// TIA Portal V20 export
FUNCTION_BLOCK "LER_SleepModeManager"   // FB184, LAD
// stored: Access Published, MemoryReserve 100, SetENOAutomatically false
   VAR_INPUT
      enable : Bool := TRUE;   // Enable sleep mode manager
      unitStatus : "LAF_typeUnitStatus";   // Unit status including stopped state and acknowledge command
      wakeUpReq : Bool;
      sleepDelay : Time;   // Idle time before sleep mode in minutes from HMI/recipe
      deepSleepDelay : Time;   // Time in sleep mode before deep sleep in minutes from HMI/recipe
   END_VAR
   VAR_OUTPUT
      sleepModeChangeReq : Bool;   // Request Unit mode change to sleep mode userMode02
      deepSleepModeChangeReq : Bool;   // Request Unit mode change to deep sleep mode userMode03
      wakeUpRecoveryRequired : Bool;
   END_VAR
   VAR
      instSleepDelay { ExternalAccessible := 'False'; ExternalVisible := 'False'; ExternalWritable := 'False'; S7_SetPoint := 'True'} : TON_TIME;
      instDeepSleepDelay { ExternalAccessible := 'False'; ExternalVisible := 'False'; ExternalWritable := 'False'; S7_SetPoint := 'True'} : TON_TIME;
      statStandbyReady { ExternalAccessible := 'False'; ExternalVisible := 'False'; ExternalWritable := 'False'} : Bool;
      statWakeUpRecoveryRequired { ExternalAccessible := 'False'; ExternalVisible := 'False'; ExternalWritable := 'False'} : Bool;
   END_VAR
   VAR_TEMP
      tempSleepDelayDone : Bool;
      tempDeepSleepDelayDone : Bool;
   END_VAR
   VAR CONSTANT
      MIN_TO_MS : LReal := 60000.0;   // Milliseconds per minute
      MAX_TIME_MIN : LReal := 35791.0;   // TIME max is about 24d20h31m23s
   END_VAR
BEGIN

REGION Network 1: Standby Ready
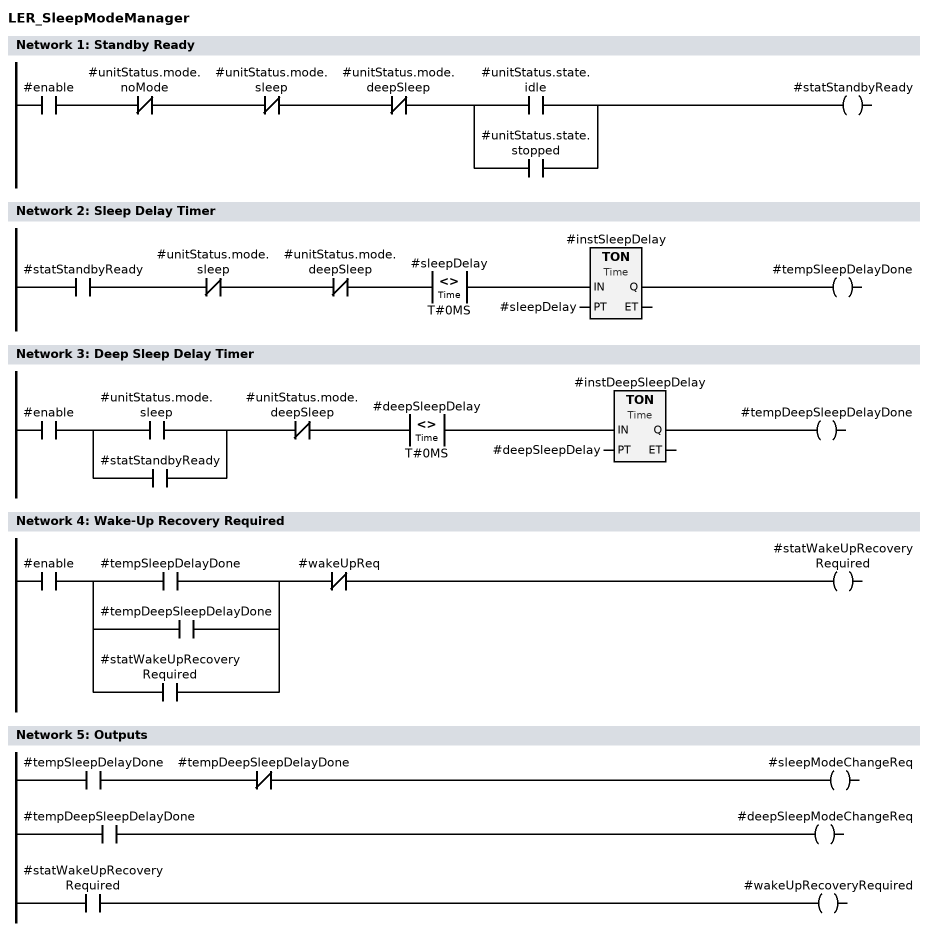
   RUNG wire#powerrail
      Contact( #enable )
      I_Contact( #unitStatus.mode.noMode )
      I_Contact( #unitStatus.mode.sleep )
      I_Contact( #unitStatus.mode.deepSleep )
      wire#w1
      Contact( #unitStatus.state.idle )
      wire#w2
      Coil( #statStandbyReady )
   END_RUNG
   RUNG wire#w1
      Contact( #unitStatus.state.stopped )
   END_RUNG wire#w2
   // the same network as SCL:
   #statStandbyReady := #enable AND NOT #unitStatus.mode.noMode AND NOT #unitStatus.mode.sleep AND NOT #unitStatus.mode.deepSleep AND (#unitStatus.state.idle OR #unitStatus.state.stopped);
END_REGION

REGION Network 2: Sleep Delay Timer
   RUNG wire#powerrail
      Contact( #statStandbyReady )
      I_Contact( #unitStatus.mode.sleep )
      I_Contact( #unitStatus.mode.deepSleep )
      { S7_Templates := "SrcType := Time" } NE_Contact(in1 := #sleepDelay, in2 := T#0MS)
      { S7_Templates := "time_type := Time" } #instSleepDelay.TON(pt := #sleepDelay, et =>)
      Coil( #tempSleepDelayDone )
   END_RUNG
   // the same network as SCL:
   #instSleepDelay(IN := #statStandbyReady AND NOT #unitStatus.mode.sleep AND NOT #unitStatus.mode.deepSleep AND (#sleepDelay <> T#0MS),   // TON
                   PT := #sleepDelay);
   #tempSleepDelayDone := #instSleepDelay.Q;
END_REGION

REGION Network 3: Deep Sleep Delay Timer
   RUNG wire#powerrail
      Contact( #enable )
      wire#w1
      Contact( #unitStatus.mode.sleep )
      wire#w2
      I_Contact( #unitStatus.mode.deepSleep )
      { S7_Templates := "SrcType := Time" } NE_Contact(in1 := #deepSleepDelay, in2 := T#0MS)
      { S7_Templates := "time_type := Time" } #instDeepSleepDelay.TON(pt := #deepSleepDelay, et =>)
      Coil( #tempDeepSleepDelayDone )
   END_RUNG
   RUNG wire#w1
      Contact( #statStandbyReady )
   END_RUNG wire#w2
   // the same network as SCL:
   #instDeepSleepDelay(IN := #enable AND (#unitStatus.mode.sleep OR #statStandbyReady) AND NOT #unitStatus.mode.deepSleep AND (#deepSleepDelay <> T#0MS),   // TON
                       PT := #deepSleepDelay);
   #tempDeepSleepDelayDone := #instDeepSleepDelay.Q;
END_REGION

REGION Network 4: Wake-Up Recovery Required
   RUNG wire#powerrail
      Contact( #enable )
      wire#w1
      Contact( #tempSleepDelayDone )
      wire#w2
      I_Contact( #wakeUpReq )
      Coil( #statWakeUpRecoveryRequired )
   END_RUNG
   RUNG wire#w1
      Contact( #tempDeepSleepDelayDone )
   END_RUNG wire#w2
   RUNG wire#w1
      Contact( #statWakeUpRecoveryRequired )
   END_RUNG wire#w2
   // the same network as SCL:
   #statWakeUpRecoveryRequired := #enable AND (#tempSleepDelayDone OR #tempDeepSleepDelayDone OR #statWakeUpRecoveryRequired) AND NOT #wakeUpReq;
END_REGION

REGION Network 5: Outputs
   RUNG wire#powerrail
      Contact( #tempSleepDelayDone )
      I_Contact( #tempDeepSleepDelayDone )
      Coil( #sleepModeChangeReq )
   END_RUNG
   RUNG wire#powerrail
      Contact( #tempDeepSleepDelayDone )
      Coil( #deepSleepModeChangeReq )
   END_RUNG
   RUNG wire#powerrail
      Contact( #statWakeUpRecoveryRequired )
      Coil( #wakeUpRecoveryRequired )
   END_RUNG
   // the same network as SCL:
   #sleepModeChangeReq := #tempSleepDelayDone AND NOT #tempDeepSleepDelayDone;
   #deepSleepModeChangeReq := #tempDeepSleepDelayDone;
   #wakeUpRecoveryRequired := #statWakeUpRecoveryRequired;
END_REGION
END_FUNCTION_BLOCK
